FUNCTION F_Log : BOOL
VAR_INPUT
	msg: STRING;
END_VAR

ADSLOGSTR(
	msgCtrlMask := ADSLOG_MSGTYPE_HINT,
	msgFmtStr := msg,
	strArg := ''
);

END_FUNCTION

(* stored: Version 1.1.0.1, ProductVersion 3.1.4024.3
   POU F_Log: Id {b4f74892-6295-4ef0-a47a-6ca0b58e2987}, SpecialFunc None *)
